// Examples of nested objects and possible variants for initialization of parent/child-relations.
FUNCTION_BLOCK FB_Struct_Nested EXTENDS FB_BA_View
VAR
	{region 'Variant 1'}
		Nested1a		: FB_NestedView				:= (View:=(iParent:=THIS^));
		Nested1b		: FB_NestedView				:= (View:=(iParent:=THIS^));
	{endregion}
	{region 'Variant 2'}
		Nested2			: FB_NestedView2			(THIS^);     
	{endregion}
END_VAR

SUPER^();

// Variant 1:
Nested1a();
Nested1b();

// Variant 2:
Nested2();

END_FUNCTION_BLOCK

(* stored: Version 1.1.0.1, ProductVersion 3.1.4024.5
   POU FB_Struct_Nested: Id {fc3d18fb-3d7e-4ba7-8d0a-fd548bfa308c}, SpecialFunc None *)
